{attribute 'linkalways'} 
{attribute 'no_explicit_call' := 'This FB is a CLASS and must be accessed using methods or properties'}
{attribute 'enable_dynamic_creation'}
FUNCTION_BLOCK _LREAL EXTENDS DatatypeBase
VAR
	localData : LREAL;
	activeData : REFERENCE TO LREAL REF= localData;
END_VAR

PROPERTY PUBLIC Address : PVOID
GET
Address := ADR(activeData);
END_GET
END_PROPERTY

METHOD PUBLIC ClearReference
VAR_INPUT
END_VAR
activeData REF= localData;
END_METHOD

METHOD PUBLIC Clone : I_Datatype
VAR
    pClone : POINTER TO _LREAL;
END_VAR
pClone := __NEW(_LREAL(InitialValue := Value));
Clone := pClone^;
END_METHOD

METHOD FB_init : BOOL
VAR_INPUT
	bInitRetains : BOOL; // if TRUE, the retain variables are initialized (warm start / cold start)
	bInCopyCode : BOOL;  // if TRUE, the instance afterwards gets moved into the copy code (online change)
	InitialValue : LREAL;
END_VAR
localData := InitialValue;
END_METHOD

PROPERTY PUBLIC IecType : T_MAXSTRING
GET
IecType := 'LREAL';
END_GET
END_PROPERTY

METHOD PUBLIC MakeReferenceTo
VAR_INPUT
	ReferenceTarget : REFERENCE TO LREAL;
END_VAR
activeData REF= ReferenceTarget;
END_METHOD

METHOD PUBLIC SerializeWith
VAR_INPUT
	Serializer : I_Serializer;
END_VAR
Serializer.AddLreal(activeData);
END_METHOD

PROPERTY PUBLIC Size : UDINT
GET
Size := SIZEOF(activeData);
END_GET
END_PROPERTY

METHOD TryDeserializeFrom : BOOL
VAR_INPUT
	Deserializer : I_Deserializer;
	Feedback : I_DeserializerFeedback;
END_VAR
TryDeserializeFrom := Deserializer.TryGetLreal(activeData, Feedback);
END_METHOD

METHOD TryMakeReferenceTo : BOOL
VAR_INPUT
	Target : I_Datatype;
END_VAR
VAR
	pTargetData : POINTER TO LREAL;
END_VAR
IF NOT (Target.IecType = IecType) THEN
	RETURN;
END_IF

pTargetData := Target.Address;
activeData REF= pTargetData^;
TryMakeReferenceTo := TRUE;
END_METHOD

PROPERTY PUBLIC Value : LREAL
GET
Value := activeData;
END_GET
SET
activeData := Value;
END_SET
END_PROPERTY

END_FUNCTION_BLOCK

(* stored: Version 1.1.0.1, ProductVersion 3.1.4024.12
   POU _LREAL: Id {cbdcb87b-08f9-0373-39c3-3d999354c82a}, SpecialFunc None
   Folder Constructor: Id {be54a52f-4d9d-0350-1d6a-4e08b8a99c1d}
   Property Address: Id {cddbdf18-21ea-0561-303c-bfe0fccf66c6}
   Get Get: Id {aa22f025-b047-0e22-33d7-7426635b118b}
   Method ClearReference: Id {a8e31a96-0fb9-0747-1447-39984eecd973}
   Method Clone: Id {f1f7eac6-2a0a-0178-3dcd-2687c83d99ee}
   Method FB_init: Id {78b86830-37f8-0c52-13f1-1480102fc30b}
   Property IecType: Id {465021d4-1ea5-06ec-2afe-3aeb73978689}
   Get Get: Id {d37b5d85-446f-0942-30b3-d9d92f7adb8f}
   Method MakeReferenceTo: Id {517ac512-77e7-0cd4-2be3-53f44615df11}
   Method SerializeWith: Id {12968aca-227b-0fcf-2321-246f5e70f092}
   Property Size: Id {c2be386e-9034-04ca-27d8-11f785e6c3dc}
   Get Get: Id {c3cbc964-b890-07d1-1812-1a24738a782c}
   Method TryDeserializeFrom: Id {4a998e4b-d930-0a87-2517-ce8b8b16faaa}
   Method TryMakeReferenceTo: Id {67d05bab-3f10-0997-256f-61ac298e826f}
   Property Value: Id {12bf45ea-abcb-00b9-2975-801a5620c575}
   Get Get: Id {57873e77-cc8b-01a8-03ba-952878a29120}
   Set Set: Id {72442890-9572-0858-33ed-928fdefe72e2} *)
